// TIA Portal V16 export
// export: Created 2021-10-05T13:40:26.4389449Z, ExportSetting None, DisplayName Totally Integrated Automation Portal, DisplayVersion V16 Update 4, DisplayName TIA Portal Version Control Interface, DisplayVersion V16 Update 2, DisplayName TIA Portal Openness, DisplayVersion V16 Update 4, DisplayName SINAMICS Startdrive Advanced, DisplayVersion V16 Update 5, DisplayName SINAMICS Startdrive G130, G150, S120, S150, SINAMICS MV, S210, DisplayVersion V16 Update 5, DisplayName SINAMICS Startdrive G110M, G120, G120C, G120D, G120P, G115D, DisplayVersion V16 Update 5, DisplayName STEP 7 Professional, DisplayVersion V16 Update 4, DisplayName STEP 7 Safety, DisplayVersion V16, DisplayName WinCC Advanced, DisplayVersion V16 Update 4
VAR_GLOBAL   // PLC tag table "AppoggiOutputs"
   MO_LampM24On AT %M420.0 : Bool;   // dosing screw M24 LED F3
   "MO_20.1" AT %M420.1 : Bool;
   "MO_20.2" AT %M420.2 : Bool;
   "MO_20.3" AT %M420.3 : Bool;
   "MO_20.4" AT %M420.4 : Bool;
   "MO_20.5" AT %M420.5 : Bool;
   "MO_20.6" AT %M420.6 : Bool;
   "MO_20.7" AT %M420.7 : Bool;
   MO_M21 AT %M421.0 : Bool;   // motor aspiration M21 on
   MO_M19 AT %M421.1 : Bool;   // rotary valve M19 on F2
   "MO_ApriDeviatoreSilosDB11-14" AT %M421.2 : Bool;   // diverter valve silo DB11-14 junction
   "MO_ChiudiDeviatoreSilosDB11-14" AT %M421.3 : Bool;   // diverter valve silo DB11-14 Dichtung
   "MO_FiltroKC13-On" AT %M421.4 : Bool;   // jetfilter KC 13 F3 on
   "MO_FiltroKC14-On" AT %M421.5 : Bool;   // jetfilter KC 14 F3 on
   MO_M23 AT %M421.6 : Bool;   // motor aspiration M23 on F3
   MO_M24 AT %M421.7 : Bool;   // dosing screw M24 on F3
   MO_SirenaSS3 AT %M422.0 : Bool;   // HORN +SS3
   "MO_DirettaSilo11-12" AT %M422.1 : Bool;   // straight to silo 11,12
   MO_M8 AT %M422.2 : Bool;   // blower M8 on
   MO_M7 AT %M422.3 : Bool;   // rotary valve M7 on
   "MO_DeviatoreSuSilos1-6" AT %M422.4 : Bool;   // Deviatore su passaggio silos 1-6
   "MO_DeviatoreSuSilos11-12" AT %M422.5 : Bool;   // Deviatore su passaggio silos 11-12
   MO_M18 AT %M422.6 : Bool;   // motor filter M 18 on
   MO_M20 AT %M422.7 : Bool;   // motor filter M 20 on F2
   MO_M1 AT %M423.0 : Bool;   // motor M1 on
   MO_M2 AT %M423.1 : Bool;   // motor M2 on
   MO_M3 AT %M423.2 : Bool;   // motor M3 on
   "MO_M4-On" AT %M423.3 : Bool;   // motor M4 on
   "MO_M5-On" AT %M423.4 : Bool;   // motor M5 on
   "MO_M6-On" AT %M423.5 : Bool;   // motor M6 on
   "MO_DirettaSilosP8-P9" AT %M423.6 : Bool;   // straight to silo P8 ,P9
   "MO_23.7" AT %M423.7 : Bool;
   MO_M22 AT %M424.0 : Bool;   // M22 rotary M22 on (P8,P9)
   MO_DirettoDeviatoreGC09 AT %M424.1 : Bool;   // diverter GC09 straight way
   "MO_24.2" AT %M424.2 : Bool;
   "MO_24.3" AT %M424.3 : Bool;
   "MO_DeviatoreSilosP8-P9" AT %M424.4 : Bool;   // diverter valve C1-GC1 (P8,P9)
   "MO_24.5" AT %M424.5 : Bool;
   "MO_24.6" AT %M424.6 : Bool;
   "MO_24.7" AT %M424.7 : Bool;
   MO_ApriDeviatoreGC05 AT %M425.0 : Bool;   // diverter GC 05
   MO_ChiudiDeviatoreGC05 AT %M425.1 : Bool;   // diverter GC 05 dichtung
   MO_ApriDeviatoreGC07 AT %M425.2 : Bool;   // diverter GC 07
   MO_ChiudiDeviatoreGC07 AT %M425.3 : Bool;   // diverter GC 07 dichtung
   MO_ApriDeviatoreGC09 AT %M425.4 : Bool;   // diverter GC 09
   MO_ChiudiDeviatoreGC09 AT %M425.5 : Bool;   // diverter GC 09 dichtung
   MO_DirettoDeviatoreGC05 AT %M425.6 : Bool;   // diverter GC05 straight way
   MO_DirettoDeviatoreGC07 AT %M425.7 : Bool;   // diverter GC07 straight way
   MO_FiltroKC01 AT %M426.0 : Bool;   // filter on DB 11
   MO_FiltroKC02 AT %M426.1 : Bool;   // filter on DB 12
   MO_FiltroKC03 AT %M426.2 : Bool;   // filter on DB 13
   MO_FiltroKC04 AT %M426.3 : Bool;   // filter on DB 14
   "MO_26.4" AT %M426.4 : Bool;
   "MO_26.5" AT %M426.5 : Bool;
   "MO_26.6" AT %M426.6 : Bool;
   "MO_26.7" AT %M426.7 : Bool;
   MO_FiltroKC12 AT %M480.0 : Bool;   // jetfilter KC 12
   "MO_SirenaSilos11-12" AT %M480.1 : Bool;   // horn silo 11,12
   "MO_LampKC12-M15-M16-On" AT %M480.2 : Bool;   // KC 12,M15,M16 on
   MO_M12 AT %M480.3 : Bool;   // M12 fluidisation blower on
   "fluidisation  solenoid valve silo 11" AT %M480.4 : Bool;   // fluidisation solenoid valve silo 11
   "fluidisation  solenoid valve silo 12" AT %M480.5 : Bool;   // fluidisation solenoid valve silo 12
   MO_M17 AT %M480.6 : Bool;   // M17 dosing screw silo 11
   MO_ValvolaM17Silo11 AT %M480.7 : Bool;   // solenoid valve silop 11 screw
   MO_M15 AT %M481.0 : Bool;   // M15 on aspiration filter
   MO_M16 AT %M481.1 : Bool;   // M16 filter motor M16 on
   MO_M11 AT %M481.2 : Bool;   // M11 dosing screw silo 12 is running
   MO_ValvolaM11Silo12 AT %M481.3 : Bool;   // GC2 solenoid valve for M11 silo 12
   MO_M14 AT %M481.4 : Bool;   // M14 conveying blower silo 11,12 on
   MO_M13 AT %M481.5 : Bool;   // M13 rotary valve on below silo 11,12
   "MO_AriaSpurgoM13Silos11-12" AT %M481.6 : Bool;   // M13 Spuelluft rotary valve
   "MO_81.7" AT %M481.7 : Bool;
END_VAR
